FUNCTION TFCalcoloOverrideDinamico : REAL
VAR_INPUT
	NUltimiTrasportiOccupati : UINT;
	Overide_Dinamico : Overide_Dinamico;
END_VAR
VAR
	i : uint;
END_VAR


FOR i:= 1 TO MAXSOGLIEOVERRIDE DO
	IF NUltimiTrasportiOccupati >= Overide_Dinamico.NTrasportiOccupati[i] THEN
		TFCalcoloOverrideDinamico := Overide_Dinamico.Override[i];
		RETURN;
	END_IF
END_FOR

END_FUNCTION

(* stored: Version 1.1.0.1, ProductVersion 3.1.4024.11
   POU TFCalcoloOverrideDinamico: Id {b9413d8f-5af3-4165-b38d-b4a42e6aa222}, SpecialFunc None *)
